Universal Robots PolyScope program: eris_v3.urp

Program eris_v2 (installation=repl_installation directory=/programs createdIn=5.16.0 lastSavedIn=5.16.0 robotSerialNumber=20185501065)
Calibrated DH parameters: a=[0.000073, -0.261994, -0.164879, -0.000046, 0.000172, 0]; d=[0.162442, 111.219294, -268.471343, 157.385991, 0.099874, 0.099634]; alpha=[1.569873, -0.003012, -0.002263, 1.572206, -1.569596, 0]; deltaTheta=[0, -0.907061, 8.327173, -1.13692, -0.000001, 0]
InitVariablesNode
Robot Program (runOnlyOnce=false)
  Script file /programs/script_code.script
    | socket_open("172.21.0.2", 8000, "abcd")
    | 
    | a = p[-0.421, -0.436, 0.1, 2.61, -1.806, -0.019]
    |  socket_send_byte(2, "abcd") socket_send_string("{", "abcd")  socket_send_byte(34, "abcd")  socket_send_string("type", "abcd")  socket_send_byte(34, "abcd")  socket_send_string(": ", "abcd")  socket_send_byte(34, "abcd")  socket_send_string("Report_state", "abcd")  socket_send_byte(34, "abcd")  socket_send_string(", ", "abcd")  socket_send_byte(34, "abcd")  socket_send_string("data", "abcd")  socket_send_byte(34, "abcd")  socket_send_string(": [{", "abcd")  socket_send_byte(34, "abcd")  socket_send_string("name", "abcd")  socket_send_byte(34, "abcd")  socket_send_string(": ", "abcd")  socket_send_byte(34, "abcd")  socket_send_string("digital_out2", "abcd")  socket_send_byte(34, "abcd")  socket_send_string(", ", "abcd")  socket_send_byte(34, "abcd")  socket_send_string("type", "abcd")  socket_send_byte(34, "abcd")  socket_send_string(": ", "abcd")  socket_send_byte(34, "abcd")  socket_send_string("String", "abcd")  socket_send_byte(34, "abcd")  socket_send_string(", ", "abcd")  socket_send_byte(34, "abcd")  socket_send_string("value", "abcd")  socket_send_byte(34, "abcd")  socket_send_string(": ", "abcd")  socket_send_byte(34, "abcd")  socket_send_string(get_digital_out(2), "abcd")  socket_send_byte(34, "abcd")  socket_send_string(", ", "abcd")  socket_send_byte(34, "abcd")  socket_send_string("global", "abcd")  socket_send_byte(34, "abcd")  socket_send_string(": true}, {", "abcd")  socket_send_byte(34, "abcd")  socket_send_string("name", "abcd")  socket_send_byte(34, "abcd")  socket_send_string(": ", "abcd")  socket_send_byte(34, "abcd")  socket_send_string("joints", "abcd")  socket_send_byte(34, "abcd")  socket_send_string(", ", "abcd")  socket_send_byte(34, "abcd")  socket_send_string("type", "abcd")  socket_send_byte(34, "abcd")  socket_send_string(": ", "abcd")  socket_send_byte(34, "abcd")  socket_send_string("String", "abcd")  socket_send_byte(34, "abcd")  socket_send_string(", ", "abcd")  socket_send_byte(34, "abcd")  socket_send_string("value", "abcd")  socket_send_byte(34, "abcd")  socket_send_string(": ", "abcd")  socket_send_byte(34, "abcd")  socket_send_string(get_actual_joint_positions(), "abcd")  socket_send_byte(34, "abcd")  socket_send_string(", ", "abcd")  socket_send_byte(34, "abcd")  socket_send_string("global", "abcd")  socket_send_byte(34, "abcd")  socket_send_string(": true}, {", "abcd")  socket_send_byte(34, "abcd")  socket_send_string("name", "abcd")  socket_send_byte(34, "abcd")  socket_send_string(": ", "abcd")  socket_send_byte(34, "abcd")  socket_send_string("digital_out6", "abcd")  socket_send_byte(34, "abcd")  socket_send_string(", ", "abcd")  socket_send_byte(34, "abcd")  socket_send_string("type", "abcd")  socket_send_byte(34, "abcd")  socket_send_string(": ", "abcd")  socket_send_byte(34, "abcd")  socket_send_string("String", "abcd")  socket_send_byte(34, "abcd")  socket_send_string(", ", "abcd")  socket_send_byte(34, "abcd")  socket_send_string("value", "abcd")  socket_send_byte(34, "abcd")  socket_send_string(": ", "abcd")  socket_send_byte(34, "abcd")  socket_send_string(get_digital_out(6), "abcd")  socket_send_byte(34, "abcd")  socket_send_string(", ", "abcd")  socket_send_byte(34, "abcd")  socket_send_string("global", "abcd")  socket_send_byte(34, "abcd")  socket_send_string(": true}, {", "abcd")  socket_send_byte(34, "abcd")  socket_send_string("name", "abcd")  socket_send_byte(34, "abcd")  socket_send_string(": ", "abcd")  socket_send_byte(34, "abcd")  socket_send_string("payload", "abcd")  socket_send_byte(34, "abcd")  socket_send_string(", ", "abcd")  socket_send_byte(34, "abcd")  socket_send_string("type", "abcd")  socket_send_byte(34, "abcd")  socket_send_string(": ", "abcd")  socket_send_byte(34, "abcd")  socket_send_string("String", "abcd")  socket_send_byte(34, "abcd")  socket_send_string(", ", "abcd")  socket_send_byte(34, "abcd")  socket_send_string("value", "abcd")  socket_send_byte(34, "abcd")  socket_send_string(": ", "abcd")  socket_send_byte(34, "abcd")  socket_send_string(get_target_payload(), "abcd")  socket_send_byte(34, "abcd")  socket_send_string(", ", "abcd")  socket_send_byte(34, "abcd")  socket_send_string("global", "abcd")  socket_send_byte(34, "abcd")  socket_send_string(": true}, {", "abcd")  socket_send_byte(34, "abcd")  socket_send_string("name", "abcd")  socket_send_byte(34, "abcd")  socket_send_string(": ", "abcd")  socket_send_byte(34, "abcd")  socket_send_string("digital_out3", "abcd")  socket_send_byte(34, "abcd")  socket_send_string(", ", "abcd")  socket_send_byte(34, "abcd")  socket_send_string("type", "abcd")  socket_send_byte(34, "abcd")  socket_send_string(": ", "abcd")  socket_send_byte(34, "abcd")  socket_send_string("String", "abcd")  socket_send_byte(34, "abcd")  socket_send_string(", ", "abcd")  socket_send_byte(34, "abcd")  socket_send_string("value", "abcd")  socket_send_byte(34, "abcd")  socket_send_string(": ", "abcd")  socket_send_byte(34, "abcd")  socket_send_string(get_digital_out(3), "abcd")  socket_send_byte(34, "abcd")  socket_send_string(", ", "abcd")  socket_send_byte(34, "abcd")  socket_send_string("global", "abcd")  socket_send_byte(34, "abcd")  socket_send_string(": true}, {", "abcd")  socket_send_byte(34, "abcd")  socket_send_string("name", "abcd")  socket_send_byte(34, "abcd")  socket_send_string(": ", "abcd")  socket_send_byte(34, "abcd")  socket_send_string("pose", "abcd")  socket_send_byte(34, "abcd")  socket_send_string(", ", "abcd")  socket_send_byte(34, "abcd")  socket_send_string("type", "abcd")  socket_send_byte(34, "abcd")  socket_send_string(": ", "abcd")  socket_send_byte(34, "abcd")  socket_send_string("String", "abcd")  socket_send_byte(34, "abcd")  socket_send_string(", ", "abcd")  socket_send_byte(34, "abcd")  socket_send_string("value", "abcd")  socket_send_byte(34, "abcd")  socket_send_string(": ", "abcd")  socket_send_byte(34, "abcd")  socket_send_string(get_actual_tcp_pose(), "abcd")  socket_send_byte(34, "abcd")  socket_send_string(", ", "abcd")  socket_send_byte(34, "abcd")  socket_send_string("global", "abcd")  socket_send_byte(34, "abcd")  socket_send_string(": true}, {", "abcd")  socket_send_byte(34, "abcd")  socket_send_string("name", "abcd")  socket_send_byte(34, "abcd")  socket_send_string(": ", "abcd")  socket_send_byte(34, "abcd")  socket_send_string("digital_out7", "abcd")  socket_send_byte(34, "abcd")  socket_send_string(", ", "abcd")  socket_send_byte(34, "abcd")  socket_send_string("type", "abcd")  socket_send_byte(34, "abcd")  socket_send_string(": ", "abcd")  socket_send_byte(34, "abcd")  socket_send_string("String", "abcd")  socket_send_byte(34, "abcd")  socket_send_string(", ", "abcd")  socket_send_byte(34, "abcd")  socket_send_string("value", "abcd")  socket_send_byte(34, "abcd")  socket_send_string(": ", "abcd")  socket_send_byte(34, "abcd")  socket_send_string(get_digital_out(7), "abcd")  socket_send_byte(34, "abcd")  socket_send_string(", ", "abcd")  socket_send_byte(34, "abcd")  socket_send_string("global", "abcd")  socket_send_byte(34, "abcd")  socket_send_string(": true}, {", "abcd")  socket_send_byte(34, "abcd")  socket_send_string("name", "abcd")  socket_send_byte(34, "abcd")  socket_send_string(": ", "abcd")  socket_send_byte(34, "abcd")  socket_send_string("digital_out0", "abcd")  socket_send_byte(34, "abcd")  socket_send_string(", ", "abcd")  socket_send_byte(34, "abcd")  socket_send_string("type", "abcd")  socket_send_byte(34, "abcd")  socket_send_string(": ", "abcd")  socket_send_byte(34, "abcd")  socket_send_string("String", "abcd")  socket_send_byte(34, "abcd")  socket_send_string(", ", "abcd")  socket_send_byte(34, "abcd")  socket_send_string("value", "abcd")  socket_send_byte(34, "abcd")  socket_send_string(": ", "abcd")  socket_send_byte(34, "abcd")  socket_send_string(get_digital_out(0), "abcd")  socket_send_byte(34, "abcd")  socket_send_string(", ", "abcd")  socket_send_byte(34, "abcd")  socket_send_string("global", "abcd")  socket_send_byte(34, "abcd")  socket_send_string(": true}, {", "abcd")  socket_send_byte(34, "abcd")  socket_send_string("name", "abcd")  socket_send_byte(34, "abcd")  socket_send_string(": ", "abcd")  socket_send_byte(34, "abcd")  socket_send_string("digital_out4", "abcd")  socket_send_byte(34, "abcd")  socket_send_string(", ", "abcd")  socket_send_byte(34, "abcd")  socket_send_string("type", "abcd")  socket_send_byte(34, "abcd")  socket_send_string(": ", "abcd")  socket_send_byte(34, "abcd")  socket_send_string("String", "abcd")  socket_send_byte(34, "abcd")  socket_send_string(", ", "abcd")  socket_send_byte(34, "abcd")  socket_send_string("value", "abcd")  socket_send_byte(34, "abcd")  socket_send_string(": ", "abcd")  socket_send_byte(34, "abcd")  socket_send_string(get_digital_out(4), "abcd")  socket_send_byte(34, "abcd")  socket_send_string(", ", "abcd")  socket_send_byte(34, "abcd")  socket_send_string("global", "abcd")  socket_send_byte(34, "abcd")  socket_send_string(": true}, {", "abcd")  socket_send_byte(34, "abcd")  socket_send_string("name", "abcd")  socket_send_byte(34, "abcd")  socket_send_string(": ", "abcd")  socket_send_byte(34, "abcd")  socket_send_string("speed", "abcd")  socket_send_byte(34, "abcd")  socket_send_string(", ", "abcd")  socket_send_byte(34, "abcd")  socket_send_string("type", "abcd")  socket_send_byte(34, "abcd")  socket_send_string(": ", "abcd")  socket_send_byte(34, "abcd")  socket_send_string("String", "abcd")  socket_send_byte(34, "abcd")  socket_send_string(", ", "abcd")  socket_send_byte(34, "abcd")  socket_send_string("value", "abcd")  socket_send_byte(34, "abcd")  socket_send_string(": ", "abcd")  socket_send_byte(34, "abcd")  socket_send_string(get_actual_joint_speeds(), "abcd")  socket_send_byte(34, "abcd")  socket_send_string(", ", "abcd")  socket_send_byte(34, "abcd")  socket_send_string("global", "abcd")  socket_send_byte(34, "abcd")  socket_send_string(": true}, {", "abcd")  socket_send_byte(34, "abcd")  socket_send_string("name", "abcd")  socket_send_byte(34, "abcd")  socket_send_string(": ", "abcd")  socket_send_byte(34, "abcd")  socket_send_string("a", "abcd")  socket_send_byte(34, "abcd")  socket_send_string(", ", "abcd")  socket_send_byte(34, "abcd")  socket_send_string("type", "abcd")  socket_send_byte(34, "abcd")  socket_send_string(": ", "abcd")  socket_send_byte(34, "abcd")  socket_send_string("String", "abcd")  socket_send_byte(34, "abcd")  socket_send_string(", ", "abcd")  socket_send_byte(34, "abcd")  socket_send_string("value", "abcd")  socket_send_byte(34, "abcd")  socket_send_string(": ", "abcd")  socket_send_byte(34, "abcd")  socket_send_string(a, "abcd")  socket_send_byte(34, "abcd")  socket_send_string(", ", "abcd")  socket_send_byte(34, "abcd")  socket_send_string("global", "abcd")  socket_send_byte(34, "abcd")  socket_send_string(": false}, {", "abcd")  socket_send_byte(34, "abcd")  socket_send_string("name", "abcd")  socket_send_byte(34, "abcd")  socket_send_string(": ", "abcd")  socket_send_byte(34, "abcd")  socket_send_string("digital_out1", "abcd")  socket_send_byte(34, "abcd")  socket_send_string(", ", "abcd")  socket_send_byte(34, "abcd")  socket_send_string("type", "abcd")  socket_send_byte(34, "abcd")  socket_send_string(": ", "abcd")  socket_send_byte(34, "abcd")  socket_send_string("String", "abcd")  socket_send_byte(34, "abcd")  socket_send_string(", ", "abcd")  socket_send_byte(34, "abcd")  socket_send_string("value", "abcd")  socket_send_byte(34, "abcd")  socket_send_string(": ", "abcd")  socket_send_byte(34, "abcd")  socket_send_string(get_digital_out(1), "abcd")  socket_send_byte(34, "abcd")  socket_send_string(", ", "abcd")  socket_send_byte(34, "abcd")  socket_send_string("global", "abcd")  socket_send_byte(34, "abcd")  socket_send_string(": true}, {", "abcd")  socket_send_byte(34, "abcd")  socket_send_string("name", "abcd")  socket_send_byte(34, "abcd")  socket_send_string(": ", "abcd")  socket_send_byte(34, "abcd")  socket_send_string("digital_out5", "abcd")  socket_send_byte(34, "abcd")  socket_send_string(", ", "abcd")  socket_send_byte(34, "abcd")  socket_send_string("type", "abcd")  socket_send_byte(34, "abcd")  socket_send_string(": ", "abcd")  socket_send_byte(34, "abcd")  socket_send_string("String", "abcd")  socket_send_byte(34, "abcd")  socket_send_string(", ", "abcd")  socket_send_byte(34, "abcd")  socket_send_string("value", "abcd")  socket_send_byte(34, "abcd")  socket_send_string(": ", "abcd")  socket_send_byte(34, "abcd")  socket_send_string(get_digital_out(5), "abcd")  socket_send_byte(34, "abcd")  socket_send_string(", ", "abcd")  socket_send_byte(34, "abcd")  socket_send_string("global", "abcd")  socket_send_byte(34, "abcd")  socket_send_string(": true}, {", "abcd")  socket_send_byte(34, "abcd")  socket_send_string("name", "abcd")  socket_send_byte(34, "abcd")  socket_send_string(": ", "abcd")  socket_send_byte(34, "abcd")  socket_send_string("force", "abcd")  socket_send_byte(34, "abcd")  socket_send_string(", ", "abcd")  socket_send_byte(34, "abcd")  socket_send_string("type", "abcd")  socket_send_byte(34, "abcd")  socket_send_string(": ", "abcd")  socket_send_byte(34, "abcd")  socket_send_string("String", "abcd")  socket_send_byte(34, "abcd")  socket_send_string(", ", "abcd")  socket_send_byte(34, "abcd")  socket_send_string("value", "abcd")  socket_send_byte(34, "abcd")  socket_send_string(": ", "abcd")  socket_send_byte(34, "abcd")  socket_send_string(get_tcp_force(), "abcd")  socket_send_byte(34, "abcd")  socket_send_string(", ", "abcd")  socket_send_byte(34, "abcd")  socket_send_string("global", "abcd")  socket_send_byte(34, "abcd")  socket_send_string(": true}], ", "abcd")  socket_send_byte(34, "abcd")  socket_send_string("id", "abcd")  socket_send_byte(34, "abcd")  socket_send_string(": 1}", "abcd")  socket_send_byte(3, "abcd")
    | movej(a, a=0.3, v=0.3)
    | 
    | b = p[-0.194, -0.6, 0.066, 2.61, -1.806, -0.019]
    | 
    | i = 0
    | while i < 5:
    |  socket_send_byte(2, "abcd") socket_send_string("{", "abcd")  socket_send_byte(34, "abcd")  socket_send_string("type", "abcd")  socket_send_byte(34, "abcd")  socket_send_string(": ", "abcd")  socket_send_byte(34, "abcd")  socket_send_string("Report_state", "abcd")  socket_send_byte(34, "abcd")  socket_send_string(", ", "abcd")  socket_send_byte(34, "abcd")  socket_send_string("data", "abcd")  socket_send_byte(34, "abcd")  socket_send_string(": [{", "abcd")  socket_send_byte(34, "abcd")  socket_send_string("name", "abcd")  socket_send_byte(34, "abcd")  socket_send_string(": ", "abcd")  socket_send_byte(34, "abcd")  socket_send_string("digital_out2", "abcd")  socket_send_byte(34, "abcd")  socket_send_string(", ", "abcd")  socket_send_byte(34, "abcd")  socket_send_string("type", "abcd")  socket_send_byte(34, "abcd")  socket_send_string(": ", "abcd")  socket_send_byte(34, "abcd")  socket_send_string("String", "abcd")  socket_send_byte(34, "abcd")  socket_send_string(", ", "abcd")  socket_send_byte(34, "abcd")  socket_send_string("value", "abcd")  socket_send_byte(34, "abcd")  socket_send_string(": ", "abcd")  socket_send_byte(34, "abcd")  socket_send_string(get_digital_out(2), "abcd")  socket_send_byte(34, "abcd")  socket_send_string(", ", "abcd")  socket_send_byte(34, "abcd")  socket_send_string("global", "abcd")  socket_send_byte(34, "abcd")  socket_send_string(": true}, {", "abcd")  socket_send_byte(34, "abcd")  socket_send_string("name", "abcd")  socket_send_byte(34, "abcd")  socket_send_string(": ", "abcd")  socket_send_byte(34, "abcd")  socket_send_string("joints", "abcd")  socket_send_byte(34, "abcd")  socket_send_string(", ", "abcd")  socket_send_byte(34, "abcd")  socket_send_string("type", "abcd")  socket_send_byte(34, "abcd")  socket_send_string(": ", "abcd")  socket_send_byte(34, "abcd")  socket_send_string("String", "abcd")  socket_send_byte(34, "abcd")  socket_send_string(", ", "abcd")  socket_send_byte(34, "abcd")  socket_send_string("value", "abcd")  socket_send_byte(34, "abcd")  socket_send_string(": ", "abcd")  socket_send_byte(34, "abcd")  socket_send_string(get_actual_joint_positions(), "abcd")  socket_send_byte(34, "abcd")  socket_send_string(", ", "abcd")  socket_send_byte(34, "abcd")  socket_send_string("global", "abcd")  socket_send_byte(34, "abcd")  socket_send_string(": true}, {", "abcd")  socket_send_byte(34, "abcd")  socket_send_string("name", "abcd")  socket_send_byte(34, "abcd")  socket_send_string(": ", "abcd")  socket_send_byte(34, "abcd")  socket_send_string("digital_out6", "abcd")  socket_send_byte(34, "abcd")  socket_send_string(", ", "abcd")  socket_send_byte(34, "abcd")  socket_send_string("type", "abcd")  socket_send_byte(34, "abcd")  socket_send_string(": ", "abcd")  socket_send_byte(34, "abcd")  socket_send_string("String", "abcd")  socket_send_byte(34, "abcd")  socket_send_string(", ", "abcd")  socket_send_byte(34, "abcd")  socket_send_string("value", "abcd")  socket_send_byte(34, "abcd")  socket_send_string(": ", "abcd")  socket_send_byte(34, "abcd")  socket_send_string(get_digital_out(6), "abcd")  socket_send_byte(34, "abcd")  socket_send_string(", ", "abcd")  socket_send_byte(34, "abcd")  socket_send_string("global", "abcd")  socket_send_byte(34, "abcd")  socket_send_string(": true}, {", "abcd")  socket_send_byte(34, "abcd")  socket_send_string("name", "abcd")  socket_send_byte(34, "abcd")  socket_send_string(": ", "abcd")  socket_send_byte(34, "abcd")  socket_send_string("payload", "abcd")  socket_send_byte(34, "abcd")  socket_send_string(", ", "abcd")  socket_send_byte(34, "abcd")  socket_send_string("type", "abcd")  socket_send_byte(34, "abcd")  socket_send_string(": ", "abcd")  socket_send_byte(34, "abcd")  socket_send_string("String", "abcd")  socket_send_byte(34, "abcd")  socket_send_string(", ", "abcd")  socket_send_byte(34, "abcd")  socket_send_string("value", "abcd")  socket_send_byte(34, "abcd")  socket_send_string(": ", "abcd")  socket_send_byte(34, "abcd")  socket_send_string(get_target_payload(), "abcd")  socket_send_byte(34, "abcd")  socket_send_string(", ", "abcd")  socket_send_byte(34, "abcd")  socket_send_string("global", "abcd")  socket_send_byte(34, "abcd")  socket_send_string(": true}, {", "abcd")  socket_send_byte(34, "abcd")  socket_send_string("name", "abcd")  socket_send_byte(34, "abcd")  socket_send_string(": ", "abcd")  socket_send_byte(34, "abcd")  socket_send_string("digital_out3", "abcd")  socket_send_byte(34, "abcd")  socket_send_string(", ", "abcd")  socket_send_byte(34, "abcd")  socket_send_string("type", "abcd")  socket_send_byte(34, "abcd")  socket_send_string(": ", "abcd")  socket_send_byte(34, "abcd")  socket_send_string("String", "abcd")  socket_send_byte(34, "abcd")  socket_send_string(", ", "abcd")  socket_send_byte(34, "abcd")  socket_send_string("value", "abcd")  socket_send_byte(34, "abcd")  socket_send_string(": ", "abcd")  socket_send_byte(34, "abcd")  socket_send_string(get_digital_out(3), "abcd")  socket_send_byte(34, "abcd")  socket_send_string(", ", "abcd")  socket_send_byte(34, "abcd")  socket_send_string("global", "abcd")  socket_send_byte(34, "abcd")  socket_send_string(": true}, {", "abcd")  socket_send_byte(34, "abcd")  socket_send_string("name", "abcd")  socket_send_byte(34, "abcd")  socket_send_string(": ", "abcd")  socket_send_byte(34, "abcd")  socket_send_string("pose", "abcd")  socket_send_byte(34, "abcd")  socket_send_string(", ", "abcd")  socket_send_byte(34, "abcd")  socket_send_string("type", "abcd")  socket_send_byte(34, "abcd")  socket_send_string(": ", "abcd")  socket_send_byte(34, "abcd")  socket_send_string("String", "abcd")  socket_send_byte(34, "abcd")  socket_send_string(", ", "abcd")  socket_send_byte(34, "abcd")  socket_send_string("value", "abcd")  socket_send_byte(34, "abcd")  socket_send_string(": ", "abcd")  socket_send_byte(34, "abcd")  socket_send_string(get_actual_tcp_pose(), "abcd")  socket_send_byte(34, "abcd")  socket_send_string(", ", "abcd")  socket_send_byte(34, "abcd")  socket_send_string("global", "abcd")  socket_send_byte(34, "abcd")  socket_send_string(": true}, {", "abcd")  socket_send_byte(34, "abcd")  socket_send_string("name", "abcd")  socket_send_byte(34, "abcd")  socket_send_string(": ", "abcd")  socket_send_byte(34, "abcd")  socket_send_string("digital_out7", "abcd")  socket_send_byte(34, "abcd")  socket_send_string(", ", "abcd")  socket_send_byte(34, "abcd")  socket_send_string("type", "abcd")  socket_send_byte(34, "abcd")  socket_send_string(": ", "abcd")  socket_send_byte(34, "abcd")  socket_send_string("String", "abcd")  socket_send_byte(34, "abcd")  socket_send_string(", ", "abcd")  socket_send_byte(34, "abcd")  socket_send_string("value", "abcd")  socket_send_byte(34, "abcd")  socket_send_string(": ", "abcd")  socket_send_byte(34, "abcd")  socket_send_string(get_digital_out(7), "abcd")  socket_send_byte(34, "abcd")  socket_send_string(", ", "abcd")  socket_send_byte(34, "abcd")  socket_send_string("global", "abcd")  socket_send_byte(34, "abcd")  socket_send_string(": true}, {", "abcd")  socket_send_byte(34, "abcd")  socket_send_string("name", "abcd")  socket_send_byte(34, "abcd")  socket_send_string(": ", "abcd")  socket_send_byte(34, "abcd")  socket_send_string("digital_out0", "abcd")  socket_send_byte(34, "abcd")  socket_send_string(", ", "abcd")  socket_send_byte(34, "abcd")  socket_send_string("type", "abcd")  socket_send_byte(34, "abcd")  socket_send_string(": ", "abcd")  socket_send_byte(34, "abcd")  socket_send_string("String", "abcd")  socket_send_byte(34, "abcd")  socket_send_string(", ", "abcd")  socket_send_byte(34, "abcd")  socket_send_string("value", "abcd")  socket_send_byte(34, "abcd")  socket_send_string(": ", "abcd")  socket_send_byte(34, "abcd")  socket_send_string(get_digital_out(0), "abcd")  socket_send_byte(34, "abcd")  socket_send_string(", ", "abcd")  socket_send_byte(34, "abcd")  socket_send_string("global", "abcd")  socket_send_byte(34, "abcd")  socket_send_string(": true}, {", "abcd")  socket_send_byte(34, "abcd")  socket_send_string("name", "abcd")  socket_send_byte(34, "abcd")  socket_send_string(": ", "abcd")  socket_send_byte(34, "abcd")  socket_send_string("digital_out4", "abcd")  socket_send_byte(34, "abcd")  socket_send_string(", ", "abcd")  socket_send_byte(34, "abcd")  socket_send_string("type", "abcd")  socket_send_byte(34, "abcd")  socket_send_string(": ", "abcd")  socket_send_byte(34, "abcd")  socket_send_string("String", "abcd")  socket_send_byte(34, "abcd")  socket_send_string(", ", "abcd")  socket_send_byte(34, "abcd")  socket_send_string("value", "abcd")  socket_send_byte(34, "abcd")  socket_send_string(": ", "abcd")  socket_send_byte(34, "abcd")  socket_send_string(get_digital_out(4), "abcd")  socket_send_byte(34, "abcd")  socket_send_string(", ", "abcd")  socket_send_byte(34, "abcd")  socket_send_string("global", "abcd")  socket_send_byte(34, "abcd")  socket_send_string(": true}, {", "abcd")  socket_send_byte(34, "abcd")  socket_send_string("name", "abcd")  socket_send_byte(34, "abcd")  socket_send_string(": ", "abcd")  socket_send_byte(34, "abcd")  socket_send_string("speed", "abcd")  socket_send_byte(34, "abcd")  socket_send_string(", ", "abcd")  socket_send_byte(34, "abcd")  socket_send_string("type", "abcd")  socket_send_byte(34, "abcd")  socket_send_string(": ", "abcd")  socket_send_byte(34, "abcd")  socket_send_string("String", "abcd")  socket_send_byte(34, "abcd")  socket_send_string(", ", "abcd")  socket_send_byte(34, "abcd")  socket_send_string("value", "abcd")  socket_send_byte(34, "abcd")  socket_send_string(": ", "abcd")  socket_send_byte(34, "abcd")  socket_send_string(get_actual_joint_speeds(), "abcd")  socket_send_byte(34, "abcd")  socket_send_string(", ", "abcd")  socket_send_byte(34, "abcd")  socket_send_string("global", "abcd")  socket_send_byte(34, "abcd")  socket_send_string(": true}, {", "abcd")  socket_send_byte(34, "abcd")  socket_send_string("name", "abcd")  socket_send_byte(34, "abcd")  socket_send_string(": ", "abcd")  socket_send_byte(34, "abcd")  socket_send_string("digital_out1", "abcd")  socket_send_byte(34, "abcd")  socket_send_string(", ", "abcd")  socket_send_byte(34, "abcd")  socket_send_string("type", "abcd")  socket_send_byte(34, "abcd")  socket_send_string(": ", "abcd")  socket_send_byte(34, "abcd")  socket_send_string("String", "abcd")  socket_send_byte(34, "abcd")  socket_send_string(", ", "abcd")  socket_send_byte(34, "abcd")  socket_send_string("value", "abcd")  socket_send_byte(34, "abcd")  socket_send_string(": ", "abcd")  socket_send_byte(34, "abcd")  socket_send_string(get_digital_out(1), "abcd")  socket_send_byte(34, "abcd")  socket_send_string(", ", "abcd")  socket_send_byte(34, "abcd")  socket_send_string("global", "abcd")  socket_send_byte(34, "abcd")  socket_send_string(": true}, {", "abcd")  socket_send_byte(34, "abcd")  socket_send_string("name", "abcd")  socket_send_byte(34, "abcd")  socket_send_string(": ", "abcd")  socket_send_byte(34, "abcd")  socket_send_string("digital_out5", "abcd")  socket_send_byte(34, "abcd")  socket_send_string(", ", "abcd")  socket_send_byte(34, "abcd")  socket_send_string("type", "abcd")  socket_send_byte(34, "abcd")  socket_send_string(": ", "abcd")  socket_send_byte(34, "abcd")  socket_send_string("String", "abcd")  socket_send_byte(34, "abcd")  socket_send_string(", ", "abcd")  socket_send_byte(34, "abcd")  socket_send_string("value", "abcd")  socket_send_byte(34, "abcd")  socket_send_string(": ", "abcd")  socket_send_byte(34, "abcd")  socket_send_string(get_digital_out(5), "abcd")  socket_send_byte(34, "abcd")  socket_send_string(", ", "abcd")  socket_send_byte(34, "abcd")  socket_send_string("global", "abcd")  socket_send_byte(34, "abcd")  socket_send_string(": true}, {", "abcd")  socket_send_byte(34, "abcd")  socket_send_string("name", "abcd")  socket_send_byte(34, "abcd")  socket_send_string(": ", "abcd")  socket_send_byte(34, "abcd")  socket_send_string("force", "abcd")  socket_send_byte(34, "abcd")  socket_send_string(", ", "abcd")  socket_send_byte(34, "abcd")  socket_send_string("type", "abcd")  socket_send_byte(34, "abcd")  socket_send_string(": ", "abcd")  socket_send_byte(34, "abcd")  socket_send_string("String", "abcd")  socket_send_byte(34, "abcd")  socket_send_string(", ", "abcd")  socket_send_byte(34, "abcd")  socket_send_string("value", "abcd")  socket_send_byte(34, "abcd")  socket_send_string(": ", "abcd")  socket_send_byte(34, "abcd")  socket_send_string(get_tcp_force(), "abcd")  socket_send_byte(34, "abcd")  socket_send_string(", ", "abcd")  socket_send_byte(34, "abcd")  socket_send_string("global", "abcd")  socket_send_byte(34, "abcd")  socket_send_string(": true}], ", "abcd")  socket_send_byte(34, "abcd")  socket_send_string("id", "abcd")  socket_send_byte(34, "abcd")  socket_send_string(": 2}", "abcd")  socket_send_byte(3, "abcd")
    |     sleep(2)
    |     i = i + 1
    | end
    | 
    | movej(b, a=0.3, v=0.3)
  Halt
